(* PLC project Unnamed, Unknown Unnamed 1 *)
(* stored: creationDateTime 2023-04-12T08:58:52, modificationDateTime 2023-04-12T08:58:52 *)

CONFIGURATION Config0
  RESOURCE Res0 ON PLC
  END_RESOURCE
END_CONFIGURATION
